{attribute 'GeneratedUsingTerminal: EM3701-0000-0016'}
{attribute addProperty BoxType "EM3701-0000-0016"}
{attribute addProperty Id "StatusAT %I*Status_E3F6A94B6ValueAT %I*INT2"}
{attribute addProperty CRC "1526095950"}
{attribute addProperty Size "8"}
TYPE AI_Inputs_5AF6604E :
STRUCT
	{attribute addProperty Name "Status"}
	Status AT %I* : Status_E3F6A94B;
	{attribute addProperty Name "Value"}
	Value AT %I* : INT;
END_STRUCT
END_TYPE

(* stored: Version 1.2.0.0, ProductVersion 3.1.4024.9
   DUT AI_Inputs_5AF6604E: Id {ad7303b6-382f-4ee0-a4ad-51ed396a6cca} *)
